FUNCTION_BLOCK L4_FMS205_F1Producir_SFC EXTENDS L1_ControllerBase_SFC
VAR_IN_OUT
	Alime			: L3_Alimentador;
	Carga		 	: L3_PickAndPlace;
	Medid			: L3_MedidorTapa;
	Induc		 	: L3_CaptadorInductivo;
	Fotoe			: L3_DetectorFotoelectrico;
	Evacu		 	: L3_Evacuador;
	Desca			: L3_PickAndPlace;
	Plato			: L3_PlatoDivisor;
	Cinta			: L3_Cinta;
END_VAR

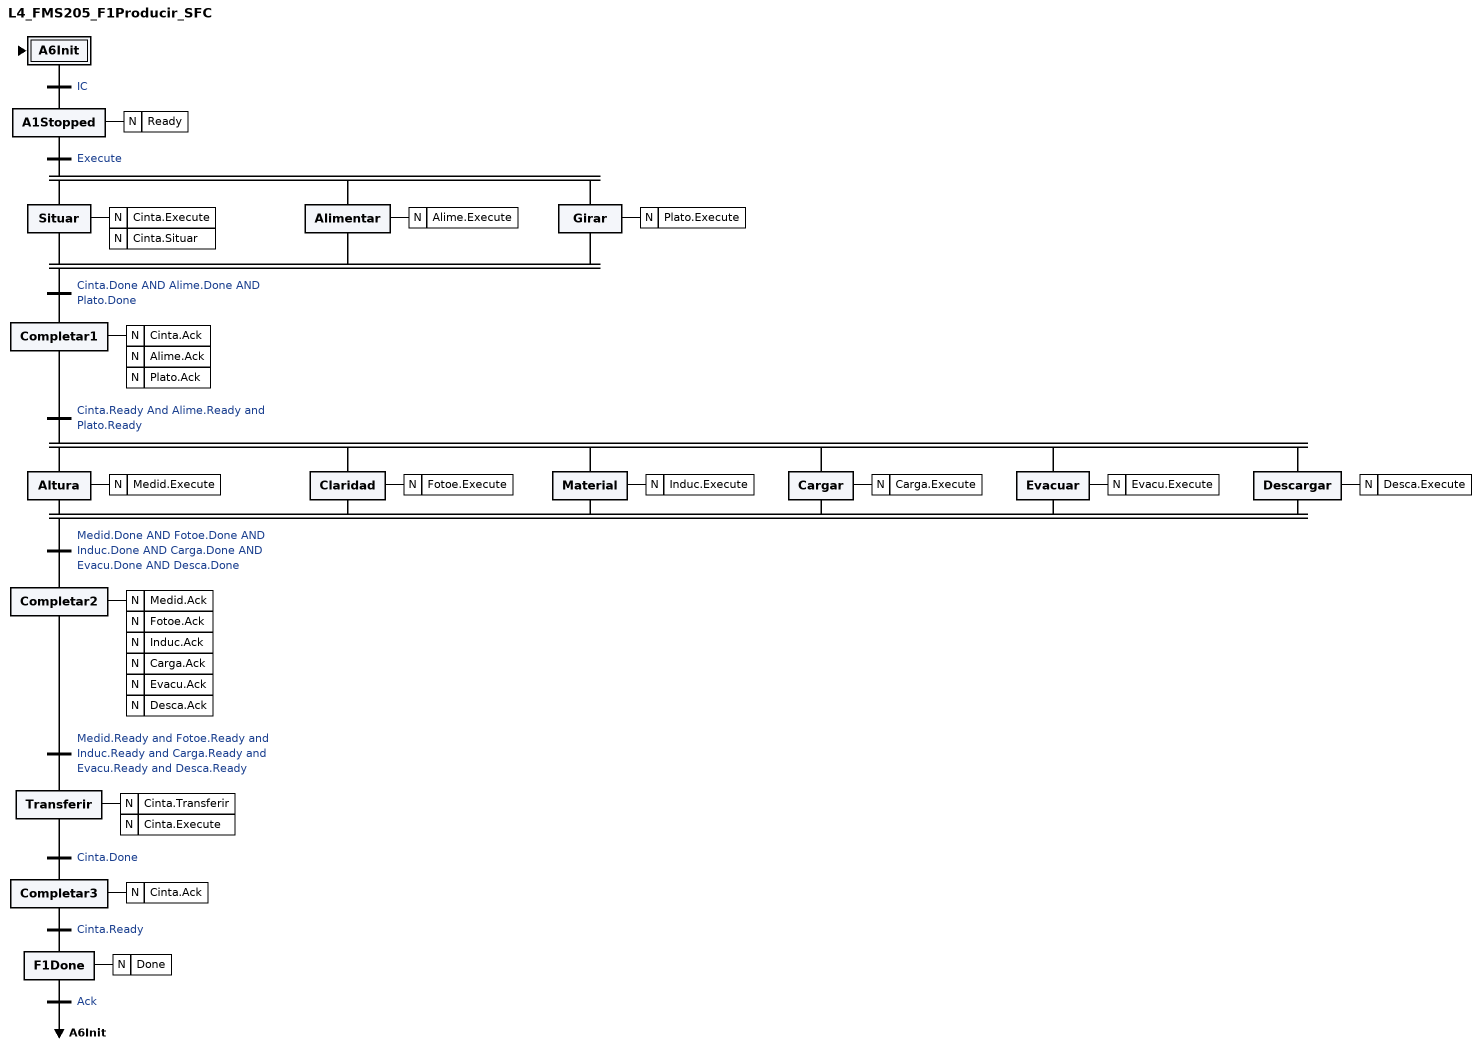
INITIAL_STEP A6Init:
END_STEP
TRANSITION FROM A6Init TO A1Stopped
    := IC;
END_TRANSITION
STEP A1Stopped:
    Ready(N);
END_STEP
TRANSITION FROM A1Stopped TO (Situar, Alimentar, Girar)
    := Execute;
END_TRANSITION
STEP Situar:
    Cinta.Execute(N);
    Cinta.Situar(N);
END_STEP
STEP Alimentar:
    Alime.Execute(N);
END_STEP
STEP Girar:
    Plato.Execute(N);
END_STEP
TRANSITION FROM (Situar, Alimentar, Girar) TO Completar1
    := Cinta.Done AND Alime.Done AND Plato.Done;
END_TRANSITION
STEP Completar1:
    Cinta.Ack(N);
    Alime.Ack(N);
    Plato.Ack(N);
END_STEP
TRANSITION FROM Completar1 TO (Altura, Claridad, Material, Cargar, Evacuar, Descargar)
    := Cinta.Ready And Alime.Ready and Plato.Ready;
END_TRANSITION
STEP Altura:
    Medid.Execute(N);
END_STEP
STEP Claridad:
    Fotoe.Execute(N);
END_STEP
STEP Material:
    Induc.Execute(N);
END_STEP
STEP Cargar:
    Carga.Execute(N);
END_STEP
STEP Evacuar:
    Evacu.Execute(N);
END_STEP
STEP Descargar:
    Desca.Execute(N);
END_STEP
TRANSITION FROM (Altura, Claridad, Material, Cargar, Evacuar, Descargar) TO Completar2
    := Medid.Done AND Fotoe.Done AND Induc.Done AND Carga.Done AND Evacu.Done AND Desca.Done;
END_TRANSITION
STEP Completar2:
    Medid.Ack(N);
    Fotoe.Ack(N);
    Induc.Ack(N);
    Carga.Ack(N);
    Evacu.Ack(N);
    Desca.Ack(N);
END_STEP
TRANSITION FROM Completar2 TO Transferir
    := Medid.Ready and Fotoe.Ready and Induc.Ready and Carga.Ready and Evacu.Ready and Desca.Ready;
END_TRANSITION
STEP Transferir:
    Cinta.Transferir(N);
    Cinta.Execute(N);
END_STEP
TRANSITION FROM Transferir TO Completar3
    := Cinta.Done;
END_TRANSITION
STEP Completar3:
    Cinta.Ack(N);
END_STEP
TRANSITION FROM Completar3 TO F1Done
    := Cinta.Ready;
END_TRANSITION
STEP F1Done:
    Done(N);
END_STEP
TRANSITION FROM F1Done TO A6Init
    := Ack;
END_TRANSITION

END_FUNCTION_BLOCK

(* stored: Version 1.1.0.1, ProductVersion 3.1.4024.11
   POU L4_FMS205_F1Producir_SFC: Id {3765931f-4c2c-4236-9e0f-0066856caec5}, SpecialFunc None *)
